// TIA Portal V17 export
// export: Created 2025-08-13T10:43:39.1705418Z, ExportSetting WithDefaults, DisplayName Totally Integrated Automation Portal, DisplayVersion V17 Update 8, DisplayName TIA Portal Openness, DisplayVersion V17 Update 8, DisplayName TIA Portal Version Control Interface, DisplayVersion V17, DisplayName SINAMICS Startdrive Advanced, DisplayVersion V17 SP2, DisplayName SINAMICS Startdrive G110M, G120, G120C, G120D, G120P, G115D, DisplayVersion V17 SP2, DisplayName SINAMICS Startdrive G130, G150, S120, S150, SINAMICS MV, S210, DisplayVersion V17 SP2, DisplayName STEP 7 Professional, DisplayVersion V17 Update 8, DisplayName STEP 7 Safety, DisplayVersion V17 Update 6, DisplayName WinCC Advanced, DisplayVersion V17 Update 8
FUNCTION_BLOCK "LaserComm_API"   // FB296, LAD
TITLE = LaserComm Communication Handling / SIS Communication Interface
{ S7_Optimized_Access := 'FALSE' }
VERSION : 2.0
// stored: AutoNumber true, IsIECCheckEnabled false, SetENOAutomatically false, UDAEnableTagReadback false
   VAR_INPUT
      iInstance_Index : Int;
      iSerial_Number : Array[1..32] of Char;
      iPart_Type : Array[1..18] of Char;
   END_VAR
   VAR DB_SPECIFIC
      sStep : Int;
      sLast_Step : Int;
      sReset : Bool;
      sLaserComm_Heart_Beat_F : Bool;
      sLaser_Heart_Beat_R : Bool;
      sHeartBeat_Dn : Bool;
      sHB_R { ExternalAccessible := 'False'; ExternalVisible := 'False'; ExternalWritable := 'False'} : Bool;
      sHB_F { ExternalAccessible := 'False'; ExternalVisible := 'False'; ExternalWritable := 'False'} : Bool;
      sLaserComm_Ready { ExternalAccessible := 'False'; ExternalVisible := 'False'; ExternalWritable := 'False'} : Bool;
      sReady_Reset : Bool;
      sLDD_Ref_Plane_Mismatch : Bool;
      sBlankResult : "LaserComm_LDD_Results";
      sBlankDDO { S7_SetPoint := 'True'} : "LaserComm_DDO";
      sData_MissMatch_Delay : IEC_TIMER;
      sStepTimeout : IEC_TIMER;
      sLaserComm_Heartbeat_Timer { S7_SetPoint := 'True'} : IEC_TIMER;
      sInstance_Inputs { S7_SetPoint := 'True'} : "API_Inputs";
      sInstance_Outputs { S7_SetPoint := 'True'} : "API_Outputs";
      sPointer : DInt;
      sHighest_Result : DInt;
   END_VAR
   VAR_TEMP
      tStep_Changed_ONS : Bool;
      tPointer : DInt;
   END_VAR
   // // sInstance_Inputs.Timeout : Timeout Value for API Job. Value set by Middleware and is dependant upon Job Function.
   VAR_TEMP   // added for the SCL form of the ladder/FBD networks
      _w1 : Bool;
      _w2 : Bool;
   END_VAR
BEGIN

REGION Network 1: Version
   // API Version
   // V1.1
   // Job Complete Flag Added to Step 30
   // Job Failed Fault Added
   // Over Pen Detection Disregarding Result Array if QA = 0
   // Move Instance Inputs and Outputs to Local Variables at Start and End of Block
   // V2
   // YLR Laser Type Supported
   // V3
   // Heart Beat Input Cleared Once Heart Beat Fault has Occurred
   // V4
   // Over Pen Bool Moved to LaserComm DB
   // Weld Mask added to LaserComm Outputs
   // Serial Number and Part Type added as inputs (Array of Chars)
   // General Tidy of Tags
   // Added Mutex
   // Added LDD Array Size constant and move to LaserComm DB register
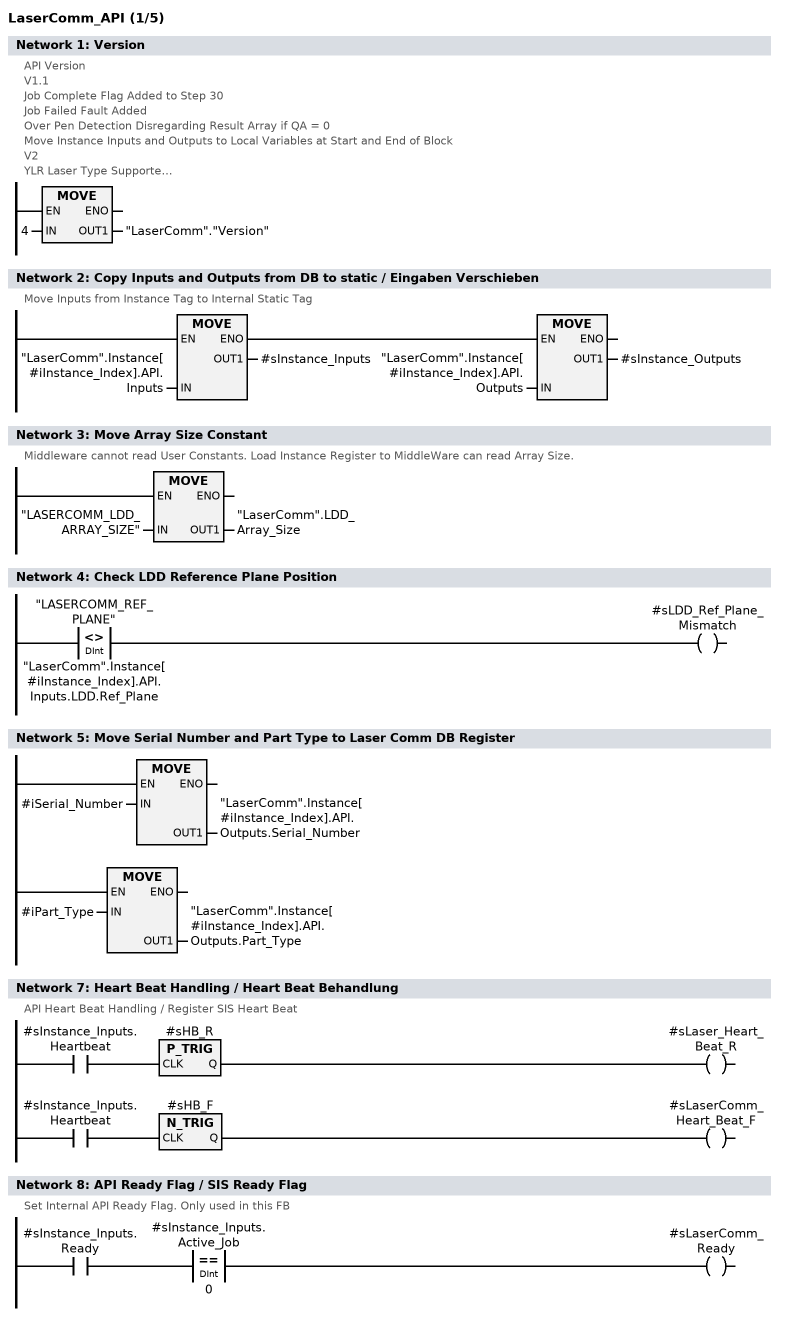
   RUNG wire#powerrail
      Move(in := 4, out1 => "LaserComm"."Version")
   END_RUNG
   // the same network as SCL:
   "LaserComm"."Version" := 4;
END_REGION

REGION Network 2: Copy Inputs and Outputs from DB to static / Eingaben Verschieben
   // Move Inputs from Instance Tag to Internal Static Tag
   RUNG wire#powerrail
      Move(in := "LaserComm".Instance[#iInstance_Index].API.Inputs, out1 => #sInstance_Inputs)
      Move(in := "LaserComm".Instance[#iInstance_Index].API.Outputs, out1 => #sInstance_Outputs)
   END_RUNG
   // the same network as SCL:
   #sInstance_Inputs := "LaserComm".Instance[#iInstance_Index].API.Inputs;
   #sInstance_Outputs := "LaserComm".Instance[#iInstance_Index].API.Outputs;
END_REGION

REGION Network 3: Move Array Size Constant
   // Middleware cannot read User Constants. Load Instance Register to MiddleWare can read Array Size.
   RUNG wire#powerrail
      Move(in := "LASERCOMM_LDD_ARRAY_SIZE", out1 => "LaserComm".LDD_Array_Size)
   END_RUNG
   // the same network as SCL:
   "LaserComm".LDD_Array_Size := "LASERCOMM_LDD_ARRAY_SIZE";
END_REGION

REGION Network 4: Check LDD Reference Plane Position
   RUNG wire#powerrail
      { S7_Templates := "SrcType := DInt" } NE_Contact(in1 := "LASERCOMM_REF_PLANE", in2 := "LaserComm".Instance[#iInstance_Index].API.Inputs.LDD.Ref_Plane)
      Coil( #sLDD_Ref_Plane_Mismatch )
   END_RUNG
   // the same network as SCL:
   #sLDD_Ref_Plane_Mismatch := "LASERCOMM_REF_PLANE" <> "LaserComm".Instance[#iInstance_Index].API.Inputs.LDD.Ref_Plane;
END_REGION

REGION Network 5: Move Serial Number and Part Type to Laser Comm DB Register
   RUNG wire#powerrail
      Move(in := #iSerial_Number, out1 => "LaserComm".Instance[#iInstance_Index].API.Outputs.Serial_Number)
   END_RUNG
   RUNG wire#powerrail
      Move(in := #iPart_Type, out1 => "LaserComm".Instance[#iInstance_Index].API.Outputs.Part_Type)
   END_RUNG
   // the same network as SCL:
   "LaserComm".Instance[#iInstance_Index].API.Outputs.Serial_Number := #iSerial_Number;
   "LaserComm".Instance[#iInstance_Index].API.Outputs.Part_Type := #iPart_Type;
END_REGION

REGION Network 6 (SCL): Over Penetration Detection / Erkennung Übermäßiger Penetration
   // Scan through the Results Array and Check for Over Penetration / Monitor QA_Results Array and look for Over Penetration Results Code
   // Monitor LDD QA Results and Check for Over Penetration
   //
   "LaserComm".Instance[#iInstance_Index].Static.OverPen_Detected := 0;

   FOR #tPointer := 0 TO "LASERCOMM_LDD_ARRAY_SIZE" DO
       IF #sInstance_Inputs.LDD.Results[#tPointer].QA <> 0 THEN
           IF #sInstance_Inputs.LDD.Results[#tPointer].Reasons.KHD.%X1 OR #sInstance_Inputs.LDD.Results[#tPointer].Reasons.KHD.%X2 THEN
               "LaserComm".Instance[#iInstance_Index].Static.OverPen_Detected := 1;
           END_IF;
       END_IF;
   END_FOR;
END_REGION

REGION Network 7: Heart Beat Handling / Heart Beat Behandlung
   // API Heart Beat Handling / Register SIS Heart Beat
   RUNG wire#powerrail
      Contact( #sInstance_Inputs.Heartbeat )
      P_Trig( #sHB_R )
      Coil( #sLaser_Heart_Beat_R )
   END_RUNG
   RUNG wire#powerrail
      Contact( #sInstance_Inputs.Heartbeat )
      N_Trig( #sHB_F )
      Coil( #sLaserComm_Heart_Beat_F )
   END_RUNG
   // the same network as SCL:
   #_w1 := #sInstance_Inputs.Heartbeat AND NOT #sHB_R;   // rising edge
   #sHB_R := #sInstance_Inputs.Heartbeat;
   #sLaser_Heart_Beat_R := #_w1;
   #_w2 := NOT #sInstance_Inputs.Heartbeat AND #sHB_F;   // falling edge
   #sHB_F := #sInstance_Inputs.Heartbeat;
   #sLaserComm_Heart_Beat_F := #_w2;
END_REGION

REGION Network 8: API Ready Flag / SIS Ready Flag
   // Set Internal API Ready Flag. Only used in this FB
   RUNG wire#powerrail
      Contact( #sInstance_Inputs.Ready )
      { S7_Templates := "SrcType := DInt" } EQ_Contact(in1 := #sInstance_Inputs.Active_Job, in2 := 0)
      Coil( #sLaserComm_Ready )
   END_RUNG
   // the same network as SCL:
   #sLaserComm_Ready := #sInstance_Inputs.Ready AND (#sInstance_Inputs.Active_Job = 0);
END_REGION

REGION Network 9: Step 0 / Schritt 0
   // Initial Step. Wait for IS Ready and Job Not Equal to 0. / Check SIS Ready, PLC Job is not 0 and PLC Start Job Is True
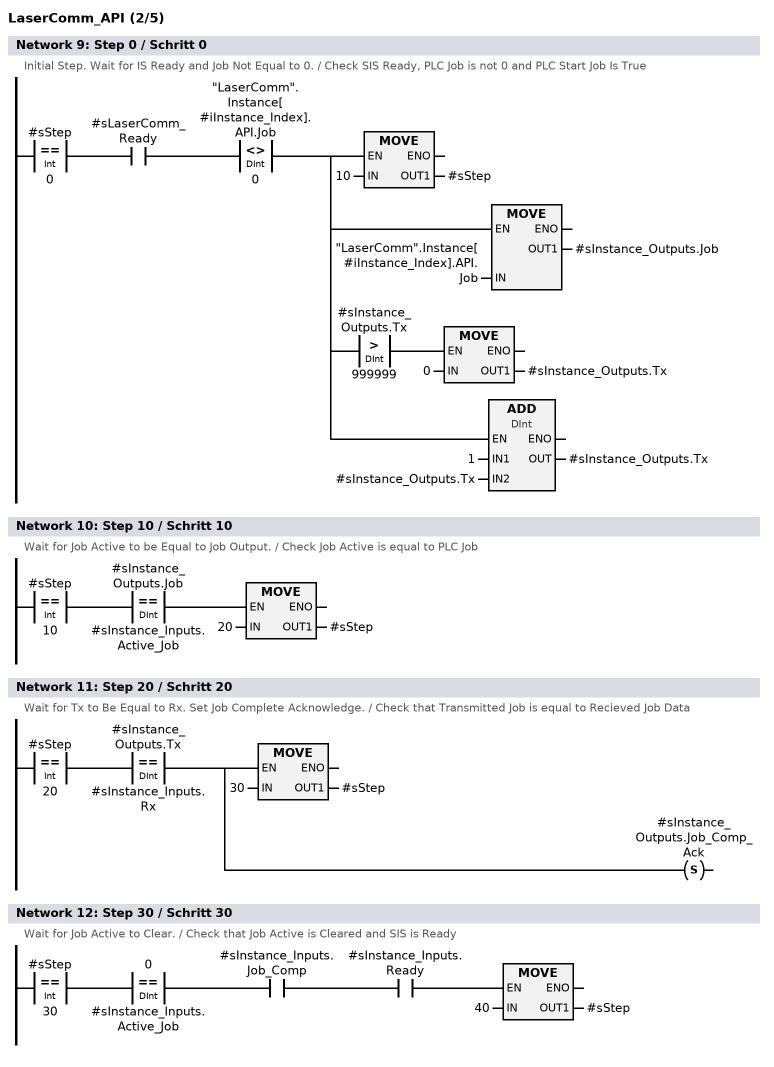
   RUNG wire#powerrail
      { S7_Templates := "SrcType := Int" } EQ_Contact(in1 := #sStep, in2 := 0)
      Contact( #sLaserComm_Ready )
      { S7_Templates := "SrcType := DInt" } NE_Contact(in1 := "LaserComm".Instance[#iInstance_Index].API.Job, in2 := 0)
      wire#w1
      { S7_GenerateENO := "TRUE" } Move(in := 10, out1 => #sStep)
   END_RUNG
   RUNG wire#w1
      { S7_GenerateENO := "TRUE" } Move(in := "LaserComm".Instance[#iInstance_Index].API.Job, out1 => #sInstance_Outputs.Job)
   END_RUNG
   RUNG wire#w1
      { S7_Templates := "SrcType := DInt" } GT_Contact(in1 := #sInstance_Outputs.Tx, in2 := 999999)
      { S7_GenerateENO := "TRUE" } Move(in := 0, out1 => #sInstance_Outputs.Tx)
   END_RUNG
   RUNG wire#w1
      { S7_Templates := "SrcType := DInt"; S7_GenerateENO := "TRUE" } Add(in1 := 1, in2 := #sInstance_Outputs.Tx, out => #sInstance_Outputs.Tx)
   END_RUNG
   // the same network as SCL:
   #_w1 := (#sStep = 0) AND #sLaserComm_Ready AND ("LaserComm".Instance[#iInstance_Index].API.Job <> 0);
   IF #_w1 THEN
       #sStep := 10;
       #sInstance_Outputs.Job := "LaserComm".Instance[#iInstance_Index].API.Job;
   END_IF;
   IF #_w1 AND (#sInstance_Outputs.Tx > 999999) THEN #sInstance_Outputs.Tx := 0; END_IF;
   IF #_w1 THEN #sInstance_Outputs.Tx := 1 + #sInstance_Outputs.Tx; END_IF;
END_REGION

REGION Network 10: Step 10 / Schritt 10
   // Wait for Job Active to be Equal to Job Output. / Check Job Active is equal to PLC Job
   RUNG wire#powerrail
      { S7_Templates := "SrcType := Int" } EQ_Contact(in1 := #sStep, in2 := 10)
      { S7_Templates := "SrcType := DInt" } EQ_Contact(in1 := #sInstance_Outputs.Job, in2 := #sInstance_Inputs.Active_Job)
      { S7_GenerateENO := "TRUE" } Move(in := 20, out1 => #sStep)
   END_RUNG
   // the same network as SCL:
   IF (#sStep = 10) AND (#sInstance_Outputs.Job = #sInstance_Inputs.Active_Job) THEN #sStep := 20; END_IF;
END_REGION

REGION Network 11: Step 20 / Schritt 20
   // Wait for Tx to Be Equal to Rx. Set Job Complete Acknowledge. / Check that Transmitted Job is equal to Recieved Job Data
   RUNG wire#powerrail
      { S7_Templates := "SrcType := Int" } EQ_Contact(in1 := #sStep, in2 := 20)
      { S7_Templates := "SrcType := DInt" } EQ_Contact(in1 := #sInstance_Outputs.Tx, in2 := #sInstance_Inputs.Rx)
      wire#w1
      { S7_GenerateENO := "TRUE" } Move(in := 30, out1 => #sStep)
   END_RUNG
   RUNG wire#w1
      S_Coil( #sInstance_Outputs.Job_Comp_Ack )
   END_RUNG
   // the same network as SCL:
   #_w1 := (#sStep = 20) AND (#sInstance_Outputs.Tx = #sInstance_Inputs.Rx);
   IF #_w1 THEN
       #sStep := 30;
       #sInstance_Outputs.Job_Comp_Ack := TRUE;
   END_IF;
END_REGION

REGION Network 12: Step 30 / Schritt 30
   // Wait for Job Active to Clear. / Check that Job Active is Cleared and SIS is Ready
   RUNG wire#powerrail
      { S7_Templates := "SrcType := Int" } EQ_Contact(in1 := #sStep, in2 := 30)
      { S7_Templates := "SrcType := DInt" } EQ_Contact(in1 := 0, in2 := #sInstance_Inputs.Active_Job)
      Contact( #sInstance_Inputs.Job_Comp )
      Contact( #sInstance_Inputs.Ready )
      { S7_GenerateENO := "TRUE" } Move(in := 40, out1 => #sStep)
   END_RUNG
   // the same network as SCL:
   IF (#sStep = 30) AND (0 = #sInstance_Inputs.Active_Job) AND #sInstance_Inputs.Job_Comp AND #sInstance_Inputs.Ready THEN
       #sStep := 40;
   END_IF;
END_REGION

REGION Network 13: Step 40 / Schritt 40
   // Reset Step
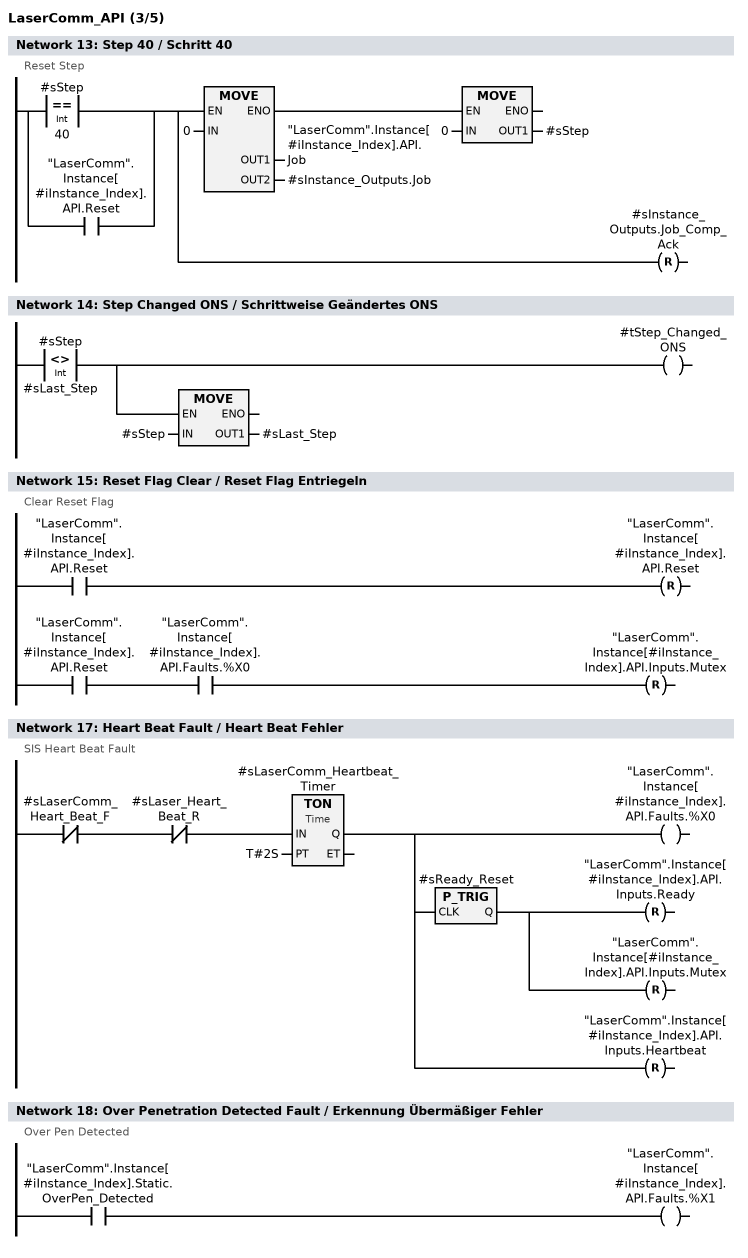
   RUNG wire#powerrail
      { S7_Templates := "SrcType := Int" } EQ_Contact(in1 := #sStep, in2 := 40)
      wire#w1
      { S7_GenerateENO := "TRUE" } Move(in := 0, out1 => "LaserComm".Instance[#iInstance_Index].API.Job, out2 => #sInstance_Outputs.Job)
      { S7_GenerateENO := "TRUE" } Move(in := 0, out1 => #sStep)
   END_RUNG
   RUNG wire#powerrail
      Contact( "LaserComm".Instance[#iInstance_Index].API.Reset )
   END_RUNG wire#w1
   RUNG wire#w1
      R_Coil( #sInstance_Outputs.Job_Comp_Ack )
   END_RUNG
   // the same network as SCL:
   // ENO of a box is taken as its EN; it also drops when the box reports an error
   #_w1 := (#sStep = 40) OR "LaserComm".Instance[#iInstance_Index].API.Reset;
   #_w2 := (#sStep = 40) OR "LaserComm".Instance[#iInstance_Index].API.Reset;
   IF #_w2 THEN
       "LaserComm".Instance[#iInstance_Index].API.Job := 0;
       #sInstance_Outputs.Job := 0;
       #sStep := 0;
   END_IF;
   IF #_w1 THEN #sInstance_Outputs.Job_Comp_Ack := FALSE; END_IF;
END_REGION

REGION Network 14: Step Changed ONS / Schrittweise Geändertes ONS
   RUNG wire#powerrail
      { S7_Templates := "SrcType := Int" } NE_Contact(in1 := #sStep, in2 := #sLast_Step)
      wire#w1
      Coil( #tStep_Changed_ONS )
   END_RUNG
   RUNG wire#w1
      { S7_GenerateENO := "TRUE" } Move(in := #sStep, out1 => #sLast_Step)
   END_RUNG
   // the same network as SCL:
   #tStep_Changed_ONS := #sStep <> #sLast_Step;
   IF #tStep_Changed_ONS THEN #sLast_Step := #sStep; END_IF;
END_REGION

REGION Network 15: Reset Flag Clear / Reset Flag Entriegeln
   // Clear Reset Flag
   RUNG wire#powerrail
      Contact( "LaserComm".Instance[#iInstance_Index].API.Reset )
      R_Coil( "LaserComm".Instance[#iInstance_Index].API.Reset )
   END_RUNG
   RUNG wire#powerrail
      Contact( "LaserComm".Instance[#iInstance_Index].API.Reset )
      Contact( "LaserComm".Instance[#iInstance_Index].API.Faults.%X0 )
      R_Coil( "LaserComm".Instance[#iInstance_Index].API.Inputs.Mutex )
   END_RUNG
   // the same network as SCL:
   IF "LaserComm".Instance[#iInstance_Index].API.Reset THEN
       "LaserComm".Instance[#iInstance_Index].API.Reset := FALSE;
   END_IF;
   IF "LaserComm".Instance[#iInstance_Index].API.Reset AND "LaserComm".Instance[#iInstance_Index].API.Faults.%X0 THEN
       "LaserComm".Instance[#iInstance_Index].API.Inputs.Mutex := FALSE;
   END_IF;
END_REGION

REGION Network 16 (SCL): Clear Results Array / Ergebnis-Array Löschen
   // Clear the Results Array

   IF #sInstance_Inputs.Clear_Results THEN
       FOR #tPointer := 0 TO "LASERCOMM_LDD_ARRAY_SIZE" DO
           "LaserComm".Instance[#iInstance_Index].API.Inputs.LDD.Results[#tPointer] := #sBlankResult;
           "LaserComm".Instance[#iInstance_Index].API.Inputs.LDD.DDO[#tPointer] := #sBlankDDO;
       END_FOR;
   END_IF;

   "LaserComm".Instance[#iInstance_Index].API.Inputs.Clear_Results := FALSE;
END_REGION

REGION Network 17: Heart Beat Fault / Heart Beat Fehler
   // SIS Heart Beat Fault
   RUNG wire#powerrail
      I_Contact( #sLaserComm_Heart_Beat_F )
      I_Contact( #sLaser_Heart_Beat_R )
      { S7_Templates := "time_type := Time" } #sLaserComm_Heartbeat_Timer.TON(pt := T#2S, et =>)
      wire#w1
      Coil( "LaserComm".Instance[#iInstance_Index].API.Faults.%X0 )
   END_RUNG
   RUNG wire#w1
      P_Trig( #sReady_Reset )
      wire#w2
      R_Coil( "LaserComm".Instance[#iInstance_Index].API.Inputs.Ready )
   END_RUNG
   RUNG wire#w2
      R_Coil( "LaserComm".Instance[#iInstance_Index].API.Inputs.Mutex )
   END_RUNG
   RUNG wire#w1
      R_Coil( "LaserComm".Instance[#iInstance_Index].API.Inputs.Heartbeat )
   END_RUNG
   // the same network as SCL:
   #sLaserComm_Heartbeat_Timer.TON(IN := NOT #sLaserComm_Heart_Beat_F AND NOT #sLaser_Heart_Beat_R, PT := T#2S);
   "LaserComm".Instance[#iInstance_Index].API.Faults.%X0 := #sLaserComm_Heartbeat_Timer.Q;
   #_w1 := #sLaserComm_Heartbeat_Timer.Q AND NOT #sReady_Reset;   // rising edge
   #sReady_Reset := #sLaserComm_Heartbeat_Timer.Q;
   IF #_w1 THEN
       "LaserComm".Instance[#iInstance_Index].API.Inputs.Ready := FALSE;
       "LaserComm".Instance[#iInstance_Index].API.Inputs.Mutex := FALSE;
   END_IF;
   IF #sLaserComm_Heartbeat_Timer.Q THEN
       "LaserComm".Instance[#iInstance_Index].API.Inputs.Heartbeat := FALSE;
   END_IF;
END_REGION

REGION Network 18: Over Penetration Detected Fault / Erkennung Übermäßiger Fehler
   // Over Pen Detected
   RUNG wire#powerrail
      Contact( "LaserComm".Instance[#iInstance_Index].Static.OverPen_Detected )
      Coil( "LaserComm".Instance[#iInstance_Index].API.Faults.%X1 )
   END_RUNG
   // the same network as SCL:
   "LaserComm".Instance[#iInstance_Index].API.Faults.%X1 := "LaserComm".Instance[#iInstance_Index].Static.OverPen_Detected;
END_REGION

REGION Network 19: Sequence Timeout Fault / Sequenz Timeout Fehler
   // SIS Command has taken too long to complete. PT Value set by SIS.
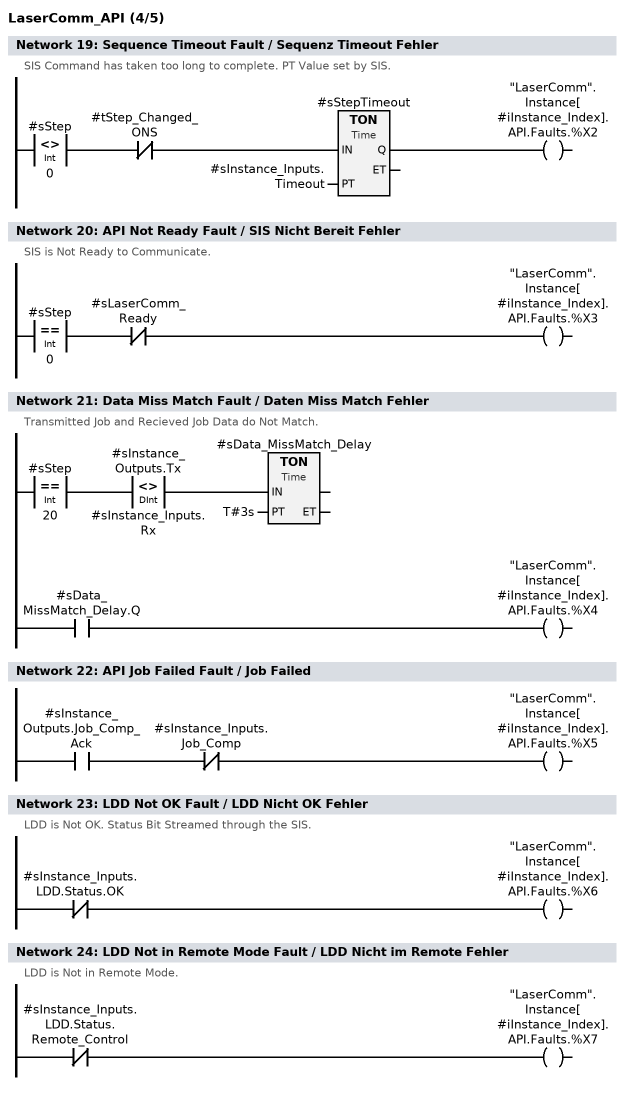
   RUNG wire#powerrail
      { S7_Templates := "SrcType := Int" } NE_Contact(in1 := #sStep, in2 := 0)
      I_Contact( #tStep_Changed_ONS )
      { S7_Templates := "time_type := Time" } #sStepTimeout.TON(pt := #sInstance_Inputs.Timeout, et =>)
      Coil( "LaserComm".Instance[#iInstance_Index].API.Faults.%X2 )
   END_RUNG
   // the same network as SCL:
   #sStepTimeout.TON(IN := (#sStep <> 0) AND NOT #tStep_Changed_ONS, PT := #sInstance_Inputs.Timeout);
   "LaserComm".Instance[#iInstance_Index].API.Faults.%X2 := #sStepTimeout.Q;
END_REGION

REGION Network 20: API Not Ready Fault / SIS Nicht Bereit Fehler
   // SIS is Not Ready to Communicate.
   RUNG wire#powerrail
      { S7_Templates := "SrcType := Int" } EQ_Contact(in1 := #sStep, in2 := 0)
      I_Contact( #sLaserComm_Ready )
      Coil( "LaserComm".Instance[#iInstance_Index].API.Faults.%X3 )
   END_RUNG
   // the same network as SCL:
   "LaserComm".Instance[#iInstance_Index].API.Faults.%X3 := (#sStep = 0) AND NOT #sLaserComm_Ready;
END_REGION

REGION Network 21: Data Miss Match Fault / Daten Miss Match Fehler
   // Transmitted Job and Recieved Job Data do Not Match.
   RUNG wire#powerrail
      { S7_Templates := "SrcType := Int" } EQ_Contact(in1 := #sStep, in2 := 20)
      { S7_Templates := "SrcType := DInt" } NE_Contact(in1 := #sInstance_Outputs.Tx, in2 := #sInstance_Inputs.Rx)
      { S7_Templates := "time_type := Time" } #sData_MissMatch_Delay.TON(pt := T#3s, et =>)
   END_RUNG
   RUNG wire#powerrail
      Contact( #sData_MissMatch_Delay.Q )
      Coil( "LaserComm".Instance[#iInstance_Index].API.Faults.%X4 )
   END_RUNG
   // the same network as SCL:
   #sData_MissMatch_Delay.TON(IN := (#sStep = 20) AND (#sInstance_Outputs.Tx <> #sInstance_Inputs.Rx),
                           PT := T#3s);
   "LaserComm".Instance[#iInstance_Index].API.Faults.%X4 := #sData_MissMatch_Delay.Q;
END_REGION

REGION Network 22: API Job Failed Fault / Job Failed
   RUNG wire#powerrail
      Contact( #sInstance_Outputs.Job_Comp_Ack )
      I_Contact( #sInstance_Inputs.Job_Comp )
      Coil( "LaserComm".Instance[#iInstance_Index].API.Faults.%X5 )
   END_RUNG
   // the same network as SCL:
   "LaserComm".Instance[#iInstance_Index].API.Faults.%X5 := #sInstance_Outputs.Job_Comp_Ack AND NOT #sInstance_Inputs.Job_Comp;
END_REGION

REGION Network 23: LDD Not OK Fault / LDD Nicht OK Fehler
   // LDD is Not OK. Status Bit Streamed through the SIS.
   RUNG wire#powerrail
      I_Contact( #sInstance_Inputs.LDD.Status.OK )
      Coil( "LaserComm".Instance[#iInstance_Index].API.Faults.%X6 )
   END_RUNG
   // the same network as SCL:
   "LaserComm".Instance[#iInstance_Index].API.Faults.%X6 := NOT #sInstance_Inputs.LDD.Status.OK;
END_REGION

REGION Network 24: LDD Not in Remote Mode Fault / LDD Nicht im Remote Fehler
   // LDD is Not in Remote Mode.
   RUNG wire#powerrail
      I_Contact( #sInstance_Inputs.LDD.Status.Remote_Control )
      Coil( "LaserComm".Instance[#iInstance_Index].API.Faults.%X7 )
   END_RUNG
   // the same network as SCL:
   "LaserComm".Instance[#iInstance_Index].API.Faults.%X7 := NOT #sInstance_Inputs.LDD.Status.Remote_Control;
END_REGION

REGION Network 25: LDD Reference Plane Mismatch Fault / LDD Nicht im Remote Fehler
   // LDD is Not in Remote Mode.
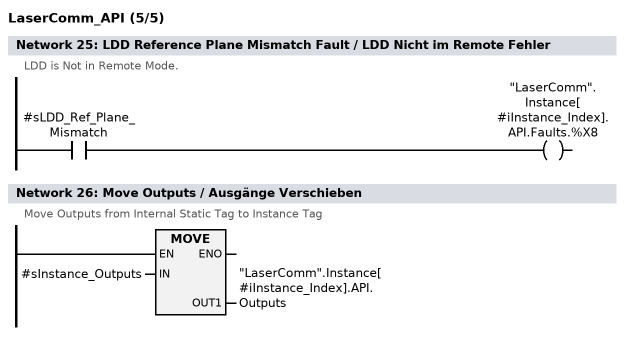
   RUNG wire#powerrail
      Contact( #sLDD_Ref_Plane_Mismatch )
      Coil( "LaserComm".Instance[#iInstance_Index].API.Faults.%X8 )
   END_RUNG
   // the same network as SCL:
   "LaserComm".Instance[#iInstance_Index].API.Faults.%X8 := #sLDD_Ref_Plane_Mismatch;
END_REGION

REGION Network 26: Move Outputs / Ausgänge Verschieben
   // Move Outputs from Internal Static Tag to Instance Tag
   RUNG wire#powerrail
      Move(in := #sInstance_Outputs, out1 => "LaserComm".Instance[#iInstance_Index].API.Outputs)
   END_RUNG
   // the same network as SCL:
   "LaserComm".Instance[#iInstance_Index].API.Outputs := #sInstance_Outputs;
END_REGION
END_FUNCTION_BLOCK
